{attribute 'qualified_only'}
{attribute 'strict'}
TYPE E_Behaviour :
(
    Pause    := 100,
    Hold     := 200,    
	Complete := 300,	
    Stop  	 := 400,    
	Abort    := 500
 );	
END_TYPE

(* stored: Version 1.1.0.1
   DUT E_Behaviour: Id {d2151b9b-4367-42a7-936d-7f67fb250d47} *)
